PROGRAM MAIN
VAR
	counter : INT := 0;
	knop : BOOL :=FALSE;
	lamp :BOOL :=FALSE;
	timer : ton;
	timer1 : ton;
	start_timer: bool;
END_VAR

//counter := counter +1; 

//IF knop THEN
//	lamp :=TRUE;
//ELSE
//	lamp:=FALSE;
//END_IF

IF gvl.StartButton THEN
	gvl.StartClamping := TRUE;
	timer1.PT := T#5S;
	timer1.IN := TRUE;
END_IF

// task clamp
IF NOT gvl.StartClamping THEN
	gvl.StateClamp := 0;
ELSE
	gvl.StateClamp := 1;
END_IF

CASE gvl.StateClamp OF 
0:
;
1:
gvl.Clamping := TRUE;
gvl.StateClamp := 2;
2:

 start_timer := TRUE;
 IF timer.Q THEN
	 gvl.StateClamp := 3;
END_IF
3:
gvl.Clamping := FALSE;
END_CASE 

// task saw
timer(IN:= start_timer, PT:= T#2000MS);

//hallo
//hallo

END_PROGRAM

(* stored: Version 1.1.0.1, ProductVersion 3.1.4024.12
   POU MAIN: Id {d02a0e1e-2859-4a94-b975-e1c9c8f0c3fe}, SpecialFunc None *)
